// SIMATIC S7-200 project (STEP 7-Micro/WIN), CPU 224 REL 02.00

SYMBOL_TABLE USER1
Start            I0.0
OUT              Q0.0
OFF              I0.1
END_SYMBOL_TABLE

ORGANIZATION_BLOCK MAIN:OB1
TITLE=PROGRAM COMMENTS
BEGIN
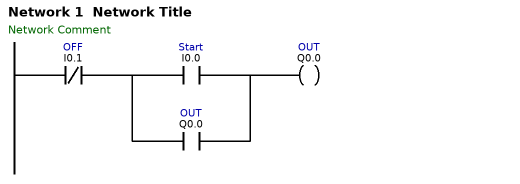
Network 1 // Network Title
// Network Comment
LDN    OFF:I0.1
LD     Start:I0.0
O      OUT:Q0.0
ALD
=      OUT:Q0.0
END_ORGANIZATION_BLOCK
